TYPE ST_GroupElements :
STRUCT
	
	
END_STRUCT
END_TYPE

(* stored: Version 1.1.0.1
   DUT ST_GroupElements: Id {40515b23-5174-0211-35e4-195f8ce597b8} *)
